FUNCTION_BLOCK FB_OuterCapillaryTubeMats EXTENDS FB_SystemContinous
VAR_INPUT
END_VAR
VAR_OUTPUT
END_VAR
VAR
	//default parameters
	localDefaultParameters : ST_OuterCapillaryTubeMatsDefaultParameters;	
	
	//pumps
	PU235 : FB_PumpGrundfosMagna3;
	PU600 : FB_PumpGrundfosMagna3;

	//valves
	ST_SV235DefaultParameters : ST_DiscreteValveDefaultParameters := (bFeedbackSignal := FALSE);
	ST_RV600DefaultParameters : ST_MixingValveDefaultParameters := (bFeedbackSignal := FALSE,aSetPointLimitsPosition := [0,100],fDefaultPosition := 0, aSetPointLimitsTemperature := [0,100], 
								fControllerAmplification := 0.265, tControllerIntegralTime := T#15S, 
								tTaskCycleTime := GlobalVariables.tTaskCycleTime_MAIN, tCtrlCycleTime := T#5S);	
	ST_RV640DefaultParameters : ST_MixingValveDefaultParameters := (bFeedbackSignal := FALSE,aSetPointLimitsPosition := [0,100],fDefaultPosition := 0, aSetPointLimitsTemperature := [0,100], 
								fControllerAmplification := 0.265, tControllerIntegralTime := T#15S, 
								tTaskCycleTime := GlobalVariables.tTaskCycleTime_MAIN, tCtrlCycleTime := T#5S);
	ST_RV660DefaultParameters : ST_MixingValveDefaultParameters := (bFeedbackSignal := FALSE,aSetPointLimitsPosition := [0,100],fDefaultPosition := 0, aSetPointLimitsTemperature := [0,100], 
								fControllerAmplification := 0.265, tControllerIntegralTime := T#15S, 
								tTaskCycleTime := GlobalVariables.tTaskCycleTime_MAIN, tCtrlCycleTime := T#5S);
	
	SV235 : FB_DiscreteValve := (ST_DefaultParameters := ST_SV235DefaultParameters);
	RV600 : FB_MixingValve := (ST_DefaultParameters := ST_RV600DefaultParameters);
	RV640 : FB_MixingValve := (ST_DefaultParameters := ST_RV640DefaultParameters); //east
	RV660 : FB_MixingValve := (ST_DefaultParameters := ST_RV660DefaultParameters); //west
	
	//sensors
	//WMZ missing
	
	//internal variables
	bSetStatusOn_PU235 : BOOL;
	bSetStatusOn_PU600 : BOOL;
	bSetStatusOn_SV235 : BOOL;	
	bSetStatusOn_RV600 : BOOL;
	bSetStatusOn_RV640 : BOOL;
	bSetStatusOn_RV660 : BOOL;
	fSetPoint_RV600 : REAL;
	fExternalTemperature_RV600 : REAL;
	nControlMode_RV600 : E_MixingValveControlMode;
	
	bStartTimer : BOOL;
	Timer : TON;
END_VAR

MAIN();
//use timer because valve has no feedback signal (75 sec)
Timer(IN := bStartTimer,
	PT := T#75S);

//pumps
//differential temperature control according to PTW6 data sheet (CHECK sign of diff temp!)
PU235(bSetStatusOnAutomatic := bSetStatusOn_PU235,
	fSetPointAutomatic := 5,
	bAlgorithmPermission := bAlgorithmPermission,
	nControlModeAutomatic := 9);
PU235.SetState_Profibus();

//use AUTO-Adapt control mode
PU600(bSetStatusOnAutomatic := bSetStatusOn_PU600,
	fSetPointAutomatic := 100,
	bAlgorithmPermission := bAlgorithmPermission,
	nControlModeAutomatic := 128);
PU600.SetState_Profibus();

//valves
SV235(bSetStatusOnAutomatic := bSetStatusOn_SV235,
	bAlgorithmPermission := bAlgorithmPermission);
SV235.SetState_BI_BO();

//RV600 uses heating mode to control inlet temperature into PWT6 (with temperature difference of 7 K of primary and secondary side)
RV600(bSetStatusOnAutomatic := bSetStatusOn_RV600,
	fSetPointAutomatic := fSetPoint-7,
	bAlgorithmPermission := bAlgorithmPermission,
	fTemperatureExternal := PU600.fTemperatureExternal,
	nControlModeAutomatic := 1);
RV600.SetState_AI_AO();

//RV640 and RV660 are alwas open
RV640(bSetStatusOnAutomatic := bSetStatusOn_RV640,
	fSetPointAutomatic := 100,
	bAlgorithmPermission := bAlgorithmPermission,
	nControlModeAutomatic := 0);
RV640.SetState_AI_AO();

RV660(bSetStatusOnAutomatic := bSetStatusOn_RV660,
	fSetPointAutomatic := 100,
	bAlgorithmPermission := bAlgorithmPermission,
	nControlModeAutomatic := 0);
RV660.SetState_AI_AO();

METHOD PROTECTED  CheckError : BOOL
VAR_INPUT
END_VAR
VAR_OUTPUT
	bError : BOOL;
END_VAR
VAR
	bError_PU235 : BOOL;
	bError_PU600 : BOOL;
	bError_SV235 : BOOL;
END_VAR
//check pumps for errors
bError_PU235 := PU235.bError;
bError_PU600 := PU600.bError;

//check valve SV235 for an error
IF SV235.bStatusOn AND PU235.bStatusOn THEN
	bError_SV235 := TRUE;
END_IF

bError := bError_PU235 OR bError_PU600 OR bError_SV235;
END_METHOD

METHOD PROTECTED  Operational : BOOL
VAR_INPUT
END_VAR
VAR_OUTPUT
	bSwitchToWorking : BOOL := FALSE;
END_VAR
bSetStatusOn_PU235 := TRUE;
bSetStatusOn_PU600 := TRUE;

IF PU235.bStatusOn AND PU600.bStatusOn THEN
	bSwitchToWorking := TRUE;
END_IF;
END_METHOD

METHOD PROTECTED  RampDown : BOOL
VAR_INPUT
END_VAR
VAR_OUTPUT
	bRampDownFinished : BOOL := FALSE;
END_VAR
bSetStatusOn_PU600 := FALSE;
bSetStatusOn_PU235 := FALSE;
bSetStatusOn_SV235 := FALSE;
bSetStatusOn_RV600 := FALSE;
bStartTimer := TRUE;

IF Timer.Q THEN
	bRampDownFinished := TRUE;
	bStartTimer := FALSE;
END_IF
END_METHOD

METHOD PROTECTED  RampUp : BOOL
VAR_INPUT
END_VAR
VAR_OUTPUT
	bRampUpFinished : BOOL := FALSE;
END_VAR
bSetStatusOn_SV235 := TRUE;
bSetStatusOn_RV600 := TRUE;
bStartTimer := TRUE;

IF Timer.Q THEN
	bRampUpFinished := TRUE;
	bStartTimer := FALSE; //resets timer
END_IF
END_METHOD

METHOD PROTECTED   SetSetPointLimits : BOOL
VAR_INPUT
END_VAR
aSetPointLimits[1] := localDefaultParameters.aSetPointLimitsTemperature[1];
aSetPointLimits[2] := localDefaultParameters.aSetPointLimitsTemperature[2];
END_METHOD

METHOD PROTECTED  Working : BOOL
VAR_INPUT
END_VAR
VAR_OUTPUT
	bSwitchToOperational : BOOL := FALSE;
END_VAR
//empty method because setpoint is passed directly to components
END_METHOD

END_FUNCTION_BLOCK

(* stored: Version 1.1.0.1, ProductVersion 3.1.4024.10
   POU FB_OuterCapillaryTubeMats: Id {f8d40369-147e-4cbe-aff1-5204bfee2138}, SpecialFunc None
   Method CheckError: Id {b5c5e5e8-42f6-4651-a2ed-f1d07717775f}
   Method Operational: Id {c5d251a1-4b82-443d-8a1b-17b15e56f92c}
   Method RampDown: Id {a23ccce8-0424-4b4c-82c7-de0b91fea1cb}
   Method RampUp: Id {a529c9d9-81e0-4127-865c-b1ad3753334d}
   Method SetSetPointLimits: Id {7fcac2fe-640f-418c-9c40-05dd5101cb8c}
   Method Working: Id {38cc873a-2ab0-456c-a4f7-7981cf3fbe46} *)
